// TIA Portal V16 export
// export: Created 2022-11-01T21:54:10.2598095Z, ExportSetting WithDefaults, DisplayName Totally Integrated Automation Portal, DisplayVersion V16, DisplayName TIA Portal Version Control Interface, DisplayVersion V16, DisplayName TIA Portal Openness, DisplayVersion V16, DisplayName SINAMICS Startdrive Advanced, DisplayVersion V16, DisplayName SINAMICS Startdrive G130, G150, S120, S150, SINAMICS MV, S210, DisplayVersion V16, DisplayName SINAMICS Startdrive G110M, G120, G120C, G120D, G120P, DisplayVersion V16, DisplayName STEP 7 Professional, DisplayVersion V16, DisplayName STEP 7 Safety, DisplayVersion V16, DisplayName WinCC Professional, DisplayVersion V16
VAR_GLOBAL   // PLC tag table "DI/O C700"
   "iH9/1_Run_Km" AT %M100.0 : Bool;
   "iH9/1_Con_Vfd" AT %M280.0 : Bool;
   "iH9/1_Run_Vfd" AT %M280.1 : Bool;
   "qH9/1_Sel_Loc/Rem" AT %M280.2 : Bool;
   "qH9/1_Sel_Km/Vfd" AT %M280.3 : Bool;
   "qH9/1_Block" AT %M280.4 : Bool;
   "qH9/1_Connect_Vfd" AT %M280.5 : Bool;
   "qH9/1_Start" AT %M280.6 : Bool;
   "iH9/2_Run_Km" AT %M280.7 : Bool;
   "iH9/2_Con_Vfd" AT %M281.0 : Bool;
   "iH9/2_Run_Vfd" AT %M281.1 : Bool;
   "qH9/2_Sel_Loc/Rem" AT %M281.2 : Bool;
   "qH9/2_Sel_Km/Vfd" AT %M281.3 : Bool;
   "qH9/2_Block" AT %M281.4 : Bool;
   "qH9/2_Connect_Vfd" AT %M281.5 : Bool;
   "qH9/2_Start" AT %M281.6 : Bool;
   "iH9/3_Run_Km" AT %M281.7 : Bool;
   "iH9/3_Con_Vfd" AT %M282.0 : Bool;
   "iH9/3_Run_Vfd" AT %M282.1 : Bool;
   "qH9/3_Sel_Loc/Rem" AT %M282.2 : Bool;
   "qH9/3_Sel_Km/Vfd" AT %M282.3 : Bool;
   "qH9/3_Block" AT %M282.4 : Bool;
   "qH9/3_Connect_Vfd" AT %M282.5 : Bool;
   "qH9/3_Start" AT %M282.6 : Bool;
   "iH9/4_Run_Km" AT %M282.7 : Bool;
   "iH9/4_Con_Vfd" AT %M283.0 : Bool;
   "iH9/4_Run_Vfd" AT %M283.1 : Bool;
   "qH9/4_Sel_Loc/Rem" AT %M283.2 : Bool;
   "qH9/4_Sel_Km/Vfd" AT %M283.3 : Bool;
   "qH9/4_Block" AT %M283.4 : Bool;
   "qH9/4_Connect_Vfd" AT %M283.5 : Bool;
   "qH9/4_Start" AT %M283.6 : Bool;
   "iH9/5_Run_Km" AT %M283.7 : Bool;
   "iH9/5_Con_Vfd" AT %M284.0 : Bool;
   "iH9/5_Run_Vfd" AT %M284.1 : Bool;
   "qH9/5_Sel_Loc/Rem" AT %M284.2 : Bool;
   "qH9/5_Sel_Km/Vfd" AT %M284.3 : Bool;
   "qH9/5_Block" AT %M284.4 : Bool;
   "qH9/5_Connect_Vfd" AT %M284.5 : Bool;
   "qH9/5_Start" AT %M284.6 : Bool;
   "iH9/6_Run_Km" AT %M284.7 : Bool;
   "iH9/6_Con_Vfd" AT %M285.0 : Bool;
   "iH9/6_Run_Vfd" AT %M285.1 : Bool;
   "qH9/6_Sel_Loc/Rem" AT %M285.2 : Bool;
   "qH9/6_Sel_Km/Vfd" AT %M285.3 : Bool;
   "qH9/6_Block" AT %M285.4 : Bool;
   "qH9/6_Connect_Vfd" AT %M285.5 : Bool;
   "qH9/6_Start" AT %M285.6 : Bool;
   "iH9/7_Run_Km" AT %M285.7 : Bool;
   "iH9/7_Con_Vfd" AT %M286.0 : Bool;
   "iH9/7_Run_Vfd" AT %M286.1 : Bool;
   "qH9/7_Sel_Loc/Rem" AT %M286.2 : Bool;
   "qH9/7_Sel_Km/Vfd" AT %M286.3 : Bool;
   "qH9/7_Block" AT %M286.4 : Bool;
   "qH9/7_Connect_Vfd" AT %M286.5 : Bool;
   "qH9/7_Start" AT %M286.6 : Bool;
   "iH9/8_Run_Km" AT %M286.7 : Bool;
   "iH9/8_Con_Vfd" AT %M287.0 : Bool;
   "iH9/8_Run_Vfd" AT %M287.1 : Bool;
   "qH9/8_Sel_Loc/Rem" AT %M287.2 : Bool;
   "qH9/8_Sel_Km/Vfd" AT %M287.3 : Bool;
   "qH9/8_Block" AT %M287.4 : Bool;
   "qH9/8_Connect_Vfd" AT %M287.5 : Bool;
   "qH9/8_Start" AT %M287.6 : Bool;
   "iH9/9_Run_Km" AT %M287.7 : Bool;
   "iH9/9_Con_Vfd" AT %M288.0 : Bool;
   "iH9/9_Run_Vfd" AT %M288.1 : Bool;
   "qH9/9_Sel_Loc/Rem" AT %M288.2 : Bool;
   "qH9/9_Sel_Km/Vfd" AT %M288.3 : Bool;
   "qH9/9_Block" AT %M288.4 : Bool;
   "qH9/9_Connect_Vfd" AT %M288.5 : Bool;
   "qH9/9_Start" AT %M288.6 : Bool;
   "iH9/10_Run_Km" AT %M288.7 : Bool;
   "iH9/10_Con_Vfd" AT %M289.0 : Bool;
   "iH9/10_Run_Vfd" AT %M289.1 : Bool;
   "qH9/10_Sel_Loc/Rem" AT %M289.2 : Bool;
   "qH9/10_Sel_Km/Vfd" AT %M289.3 : Bool;
   "qH9/10_Block" AT %M289.4 : Bool;
   "qH9/10_Connect_Vfd" AT %M289.5 : Bool;
   "qH9/10_Start" AT %M289.6 : Bool;
   "iH701/1_Run_Km" AT %M289.7 : Bool;
   "iH701/1_Con_Vfd" AT %M290.0 : Bool;
   "iH701/1_Run_Vfd" AT %M290.1 : Bool;
   "qH701/1_Sel_Loc/Rem" AT %M290.2 : Bool;
   "qH701/1_Sel_Km/Vfd" AT %M290.3 : Bool;
   "qH701/1_Block" AT %M290.4 : Bool;
   "qH701/1_Connect_Vfd" AT %M290.5 : Bool;
   "qH701/1_Start" AT %M290.6 : Bool;
   "iH701/2_Run_Km" AT %M290.7 : Bool;
   "iH701/2_Con_Vfd" AT %M291.0 : Bool;
   "iH701/2_Run_Vfd" AT %M291.1 : Bool;
   "qH701/2_Sel_Loc/Rem" AT %M291.2 : Bool;
   "qH701/2_Sel_Km/Vfd" AT %M291.3 : Bool;
   "qH701/2_Block" AT %M291.4 : Bool;
   "qH701/2_Connect_Vfd" AT %M291.5 : Bool;
   "qH701/2_Start" AT %M291.6 : Bool;
   "iH701/3_Run_Km" AT %M291.7 : Bool;
   "iH701/3_Con_Vfd" AT %M292.0 : Bool;
   "iH701/3_Run_Vfd" AT %M292.1 : Bool;
   "qH701/3_Sel_Loc/Rem" AT %M292.2 : Bool;
   "qH701/3_Sel_Km/Vfd" AT %M292.3 : Bool;
   "qH701/3_Block" AT %M292.4 : Bool;
   "qH701/3_Connect_Vfd" AT %M292.5 : Bool;
   "qH701/3_Start" AT %M292.6 : Bool;
   "iH701/4_Run_Km" AT %M292.7 : Bool;
   "iH701/4_Con_Vfd" AT %M293.0 : Bool;
   "iH701/4_Run_Vfd" AT %M293.1 : Bool;
   "qH701/4_Sel_Loc/Rem" AT %M293.2 : Bool;
   "qH701/4_Sel_Km/Vfd" AT %M293.3 : Bool;
   "qH701/4_Block" AT %M293.4 : Bool;
   "qH701/4_Connect_Vfd" AT %M293.5 : Bool;
   "qH701/4_Start" AT %M293.6 : Bool;
   "iH701/5_Run_Km" AT %M293.7 : Bool;
   "iH701/5_Con_Vfd" AT %M294.0 : Bool;
   "iH701/5_Run_Vfd" AT %M294.1 : Bool;
   "qH701/5_Sel_Loc/Rem" AT %M294.2 : Bool;
   "qH701/5_Sel_Km/Vfd" AT %M294.3 : Bool;
   "qH701/5_Block" AT %M294.4 : Bool;
   "qH701/5_Connect_Vfd" AT %M294.5 : Bool;
   "qH701/5_Start" AT %M294.6 : Bool;
   iUV701_Opn AT %M294.7 : Bool;
   iUV701_Cls AT %M295.0 : Bool;
   qUV701 AT %M295.1 : Bool;
   iUV702_Opn AT %M295.2 : Bool;
   iUV702_Cls AT %M295.3 : Bool;
   qUV702 AT %M295.4 : Bool;
   iUV703_Opn AT %M295.5 : Bool;
   iUV703_Cls AT %M295.6 : Bool;
   qUV703 AT %M295.7 : Bool;
   iUV704_Opn AT %M296.0 : Bool;
   iUV704_Cls AT %M296.1 : Bool;
   qUV704 AT %M296.2 : Bool;
   iUV705_Opn AT %M296.3 : Bool;
   iUV705_Cls AT %M296.4 : Bool;
   qUV705 AT %M296.5 : Bool;
   iUV706_Opn AT %M296.6 : Bool;
   iUV706_Cls AT %M296.7 : Bool;
   qUV706 AT %M297.0 : Bool;
   iUV707_Opn AT %M297.1 : Bool;
   iUV707_Cls AT %M297.2 : Bool;
   qUV707 AT %M297.3 : Bool;
   iUV708_Opn AT %M297.4 : Bool;
   iUV708_Cls AT %M297.5 : Bool;
   qUV708 AT %M297.6 : Bool;
   iUV709_Opn AT %M297.7 : Bool;
   iUV709_Cls AT %M298.0 : Bool;
   qUV709 AT %M298.1 : Bool;
END_VAR
